// TwinCAT 3 PLC project PLC2
// ProgramVersion: 3.1.4023.0
// libraries:
//   Tc2_Standard, * (Beckhoff Automation GmbH)
//   Tc2_System, * (Beckhoff Automation GmbH)
//   Tc2_Utilities, * (Beckhoff Automation GmbH)
//   Tc3_Database, * (Beckhoff Automation GmbH)
//   Tc3_EventLogger, * (Beckhoff Automation GmbH)
//   Tc3_Module, * (Beckhoff Automation GmbH)
// project tree:
//   / PlcTask.TcTTO, PlcUpdateData.TcTTO
//   POUs/ AdvUpdateData.TcPOU, Simulation.TcPOU
// real-time tasks:
//   TASK PlcTask: cycle T#100us, priority 20, ADS port 350
//   TASK PlcUpdateData: cycle T#100us, priority 21, ADS port 351

CONFIGURATION PLC2
    RESOURCE PLC ON TwinCAT3
        TASK PlcTask(INTERVAL := T#100us, PRIORITY := 20);
        TASK PlcUpdateData(INTERVAL := T#100us, PRIORITY := 21);
        PROGRAM Simulation WITH PlcTask : Simulation;
        PROGRAM AdvUpdateData WITH PlcUpdateData : AdvUpdateData;
    END_RESOURCE
END_CONFIGURATION

// ---- POUs/Simulation.TcPOU
PROGRAM Simulation
VAR
	rSpeed: REAL := 0;
	rPos: REAL := 0;
	bPulse: BOOL := TRUE;
	fbTon: TON;
END_VAR

fbTon(IN := NOT fbTon.Q, PT:= T#1S);
IF (fbTon.Q) THEN
	IF (rSpeed < 100) THEN
		rSpeed := rSpeed + 1.1;
	ELSE 
		rSpeed := 0;
	END_IF
	IF (rPos < 100) THEN
		rPos := rPos + 1;
	ELSE 
		rPos := 0;
	END_IF
	bPulse := NOT bPulse;
END_IF

END_PROGRAM

// ---- POUs/AdvUpdateData.TcPOU
PROGRAM AdvUpdateData
VAR
	fbSqlDatabase : FB_SQLDatabaseEvt(sNetID := '', tTimeout := T#5S);
	fbSqlCommand : FB_SQLCommandEvt(sNetID := '', tTimeout := T#5S);
	myDBID: UDINT := 1;
	sTableName: STRING := 'Data';
	sCmd: STRING(1000);
	bConnected: BOOL;

	tcMessage1 : I_TcMessage;
	tcMessage2 : I_TcMessage;
	tcMessage3 : I_TcMessage;

	systime: GETSYSTEMTIME;
	currentTime: T_FILETIME;
	timestring: string;
	iId: LINT := 1;
	
	bFirstScan: BOOL := TRUE;
	bExecute: BOOL;
	fbTon: TON;
	iLapse: USINT := 0;
	
	temp:int;
END_VAR

IF (bFirstScan) THEN
	IF fbSqlDatabase.Connect(myDBID) THEN
		bFirstScan := FALSE;
		IF fbSqlDatabase.bError THEN
			tcMessage1:= fbSqlDatabase.ipTcResult;
			bFirstScan:= TRUE;
		END_IF
	END_IF
END_IF

fbTon(IN:= NOT fbTon.Q, PT:= T#1S);
IF fbTon.Q THEN
	bExecute:= TRUE;
	systime(timeLoDW => currentTime.dwLowDateTime, timeHiDW => currentTime.dwHighDateTime);
END_IF

IF bExecute AND NOT bFirstScan THEN	
	CASE iLapse OF
		0: 
			CreateDeleteAll();
		1: 
			CreateInsert();
		2: 
			CreateUpdate();
	END_CASE
	
	IF fbSqlDatabase.CreateCmd(ADR(fbSqlCommand)) THEN
		IF fbSqlDatabase.bError THEN
			tcMessage2:= fbSqlDatabase.ipTcResult;
		END_IF
	END_IF
	
	IF fbSQLCommand.Execute(ADR(sCmd), LEN(sCmd)) THEN
		IF fbSQLCommand.bError THEN
			tcMessage3 := fbSQLCommand.ipTcResult;
		END_IF
		
		IF iLapse<>0 THEN
			iId := iId + 1;
			IF iId > 10 THEN
				iId := 1;
				iLapse := 2; 
			END_IF
		ELSE
			iLapse:=1;
		END_IF
		bExecute:= FALSE;
	END_IF
END_IF

ACTION CreateDeleteAll:
sCmd:= 'DELETE FROM ';
sCmd:= concat(sCmd, sTableName);
END_ACTION

ACTION CreateInsert:
sCmd := 'INSERT INTO ';
sCmd := concat(sCmd, sTableName);
sCmd := concat(sCmd, '( Id, Sync, Timestamp, Speed, Pos, Pulse) VALUES ( ');
sCmd := concat(sCmd, LINT_TO_STRING(iId));
sCmd := concat(sCmd, ',');
sCmd := concat(sCmd, BOOL_TO_STRING(FALSE));
sCmd := concat(sCmd, ',$'');
timestring:= DT_TO_STRING(FILETIME_TO_DT(currentTime));
timestring:= delete(timestring, 3, 1);
timestring:= replace(timestring, ' ', 1, 11);
sCmd := concat(sCmd, timestring);
sCmd := concat(sCmd, '$',');
sCmd := concat(sCmd, LREAL_TO_STRING(Simulation.rSpeed));
sCmd := concat(sCmd, ',');
sCmd := concat(sCmd, LREAL_TO_STRING(Simulation.rPos));
sCmd := concat(sCmd, ',');
sCmd := concat(sCmd, BOOL_TO_STRING(Simulation.bPulse));
sCmd := concat(sCmd, ')');
END_ACTION

ACTION CreateUpdate:
sCmd := 'UPDATE ';
sCmd := concat(sCmd, sTableName);
sCmd := concat(sCmd, ' SET Timestamp=$'');
timestring:= DT_TO_STRING(FILETIME_TO_DT(currentTime));
timestring:= delete(timestring, 3, 1);
timestring:= replace(timestring, ' ', 1, 11);
sCmd := concat(sCmd, timestring);
sCmd := concat(sCmd, '$', Speed=');
sCmd := concat(sCmd, LREAL_TO_STRING(Simulation.rSpeed));
sCmd := concat(sCmd, ', Pos=');
sCmd := concat(sCmd, LREAL_TO_STRING(Simulation.rPos));
sCmd := concat(sCmd, ', Pulse=');
sCmd := concat(sCmd, BOOL_TO_STRING(Simulation.bPulse));
sCmd := concat(sCmd, ', Sync=');
sCmd := concat(sCmd, BOOL_TO_STRING(FALSE));
sCmd := concat(sCmd, ' WHERE Id=');
sCmd := concat(sCmd, LINT_TO_STRING(iId));
END_ACTION

END_PROGRAM
